PROGRAM prgEM
VAR
	fbKBusState		: FB_K_Bus_State;
	fbEM1			: FB_EM_Beckhoff_KL3403;
	fbEM2			: FB_EM_Beckhoff_KL3403;
	fbEM3			: FB_EM_Beckhoff_KL3403;
	fbEM4			: FB_EM_Beckhoff_KL3403;
	fbEM5			: FB_EM_Beckhoff_KL3403;
	
	wDataL1, wDataL2, wDataL3   AT%I* : WORD;
	bySBL1, bySBL2, bySBL3      AT%I* : BYTE;
	byCBL1, byCBL2, byCBL3      AT%Q*       : BYTE;
	iDataOutL1, iDataOutL2, iDataOutL3  AT%Q* : INT;
	
	fbEM6			: FB_EM_Beckhoff_KL3403;
	fbEM7			: FB_EM_Beckhoff_KL3403;
	fbEM8			: FB_EM_Beckhoff_KL3403;
	fbGrid			: FB_Grid_Power_Ext_Input;			//{#lynus.ag#()}
	lrPowerEM1		: LREAL;							//{#lynus.ag#()}
	lrPowerEM2		: LREAL;							//{#lynus.ag#()}
	lrPowerEM3		: LREAL;							//{#lynus.ag#()}
	lrPowerEM4		: LREAL;							//{#lynus.ag#()}
	lrPowerEM5		: LREAL;							//{#lynus.ag#()}
	lrPowerEM5_1	: LREAL;							//{#lynus.ag#()}
	lrPowerEM5_2	: LREAL;							//{#lynus.ag#()}
	lrPowerEM5_3	: LREAL;							//{#lynus.ag#()}
	lrPowerEM6		: LREAL;							//{#lynus.ag#()}
	lrPowerEM6_1	: LREAL;							//{#lynus.ag#()}
	lrPowerEM6_2	: LREAL;							//{#lynus.ag#()}
	lrPowerEM6_3	: LREAL;							//{#lynus.ag#()}
	lrPowerEM7		: LREAL;							//{#lynus.ag#()}
	lrPowerEM7_1	: LREAL;							//{#lynus.ag#()}
	lrPowerEM7_2	: LREAL;							//{#lynus.ag#()}
	lrPowerEM7_3	: LREAL;							//{#lynus.ag#()}
	lrPowerEM8		: LREAL;							//{#lynus.ag#()}
	lrPowerEM8_1	: LREAL;							//{#lynus.ag#()}
	lrPowerEM8_2	: LREAL;							//{#lynus.ag#()}
	lrPowerEM8_3	: LREAL;							//{#lynus.ag#()}
	lrCounterEM5	: LREAL;							//{#lynus.ag#()}
	lrCounterEM6	: LREAL;							//{#lynus.ag#()}
	lrCounterEM7	: LREAL;							//{#lynus.ag#()}
	lrCounterEM8	: LREAL;							//{#lynus.ag#()}
	
	lrCurrent_EM5_1 : LREAL;							//{#lynus.ag#()}
	lrCurrent_EM5_2 : LREAL;							//{#lynus.ag#()}
	lrCurrent_EM5_3 : LREAL;							//{#lynus.ag#()}
	lrCurrent_EM6_1 : LREAL;							//{#lynus.ag#()}
	lrCurrent_EM6_2 : LREAL;							//{#lynus.ag#()}
	lrCurrent_EM6_3 : LREAL;							//{#lynus.ag#()}
	lrCurrent_EM7_1 : LREAL;							//{#lynus.ag#()}
	lrCurrent_EM7_2 : LREAL;							//{#lynus.ag#()}
	lrCurrent_EM7_3 : LREAL;							//{#lynus.ag#()}
	lrCurrent_EM8_1 : LREAL;							//{#lynus.ag#()}
	lrCurrent_EM8_2 : LREAL;							//{#lynus.ag#()}
	lrCurrent_EM8_3 : LREAL;							//{#lynus.ag#()}
END_VAR

fbKBusState(uiKBusState_OUT=> );


//UV1	
fbEM1(
	bEnable:= TRUE, 
	bChannel1Invers:= TRUE,
	bChannel2Invers:= TRUE,
	bChannel3Invers:= TRUE,
	uiCurrentTransformerRatioL1:= 400, 
	uiCurrentTransformerRatioL2:= 400, 
	uiCurrentTransformerRatioL3:= 400, 
	uiKBusState_IN:= fbKBusState.uiKBusState_OUT, 
	stDataEMPower=> , 
	stDataEMCounter=> , 
	stDataEMPowerRealTime=> , 
	stDataEMCounterRealTime=> , 
	diNrOfEM_OUT=> );

lrPowerEM1 := fbEM1.stDataEMPower.lrPowerTotal;

//UV2	
fbEM2(
	bEnable:= TRUE, 
	bChannel1Invers:= TRUE,
	bChannel2Invers:= TRUE,
	bChannel3Invers:= TRUE,
	uiCurrentTransformerRatioL1:= 400, 
	uiCurrentTransformerRatioL2:= 400, 
	uiCurrentTransformerRatioL3:= 400, 
	uiKBusState_IN:= fbKBusState.uiKBusState_OUT, 
	stDataEMPower=> , 
	stDataEMCounter=> , 
	stDataEMPowerRealTime=> , 
	stDataEMCounterRealTime=> , 
	diNrOfEM_OUT=> );

lrPowerEM2 := fbEM2.stDataEMPower.lrPowerTotal;

//UV3	
fbEM3(
	bEnable:= TRUE, 
	bChannel1Invers:= TRUE,
	bChannel2Invers:= TRUE,
	bChannel3Invers:= TRUE,
	uiCurrentTransformerRatioL1:= 400, 
	uiCurrentTransformerRatioL2:= 400, 
	uiCurrentTransformerRatioL3:= 400, 
	uiKBusState_IN:= fbKBusState.uiKBusState_OUT, 
	stDataEMPower=> , 
	stDataEMCounter=> , 
	stDataEMPowerRealTime=> , 
	stDataEMCounterRealTime=> , 
	diNrOfEM_OUT=> );

lrPowerEM3 := fbEM3.stDataEMPower.lrPowerTotal;	
	
//UV4	
fbEM4(
	bEnable:= TRUE, 
	bChannel1Invers:= TRUE,
	bChannel2Invers:= TRUE,
	bChannel3Invers:= TRUE,
	uiCurrentTransformerRatioL1:= 400, 
	uiCurrentTransformerRatioL2:= 400, 
	uiCurrentTransformerRatioL3:= 400, 
	uiKBusState_IN:= fbKBusState.uiKBusState_OUT, 
	stDataEMPower=> , 
	stDataEMCounter=> , 
	stDataEMPowerRealTime=> , 
	stDataEMCounterRealTime=> , 
	diNrOfEM_OUT=> );

lrPowerEM4 := fbEM4.stDataEMPower.lrPowerTotal;	

//UV5	
fbEM5(
	bEnable:= TRUE, 
	bChannel1Invers:= TRUE,
	bChannel2Invers:= TRUE,
	bChannel3Invers:= TRUE,
	uiCurrentTransformerRatioL1:= 400, 
	uiCurrentTransformerRatioL2:= 400, 
	uiCurrentTransformerRatioL3:= 400, 
	uiKBusState_IN:= fbKBusState.uiKBusState_OUT, 
	stDataEMPower=> , 
	stDataEMCounter=> , 
	stDataEMPowerRealTime=> , 
	stDataEMCounterRealTime=> , 
	diNrOfEM_OUT=> );

lrPowerEM5 := fbEM5.stDataEMPower.lrPowerTotal;	
	lrCounterEM5 := fbEM5.stDataEMCounter.lrTotalCounterEnergy_Consumption;	
		lrPowerEM5_1 := fbEM5.stDataEMPower.lrPowerL1;
			lrPowerEM5_2 := fbEM5.stDataEMPower.lrPowerL2;
				lrPowerEM5_3 := fbEM5.stDataEMPower.lrPowerL3;
					lrCurrent_EM5_1 := fbEM5.stDataEMPower.lrCurrentL1;
						lrCurrent_EM5_2 := fbEM5.stDataEMPower.lrCurrentL2;
							lrCurrent_EM5_3 := fbEM5.stDataEMPower.lrCurrentL3;
	
//UV6
fbEM6(
	bEnable:= TRUE, 
	bChannel1Invers:= TRUE,
	bChannel2Invers:= TRUE,
	bChannel3Invers:= TRUE,
	uiCurrentTransformerRatioL1:= 400, 
	uiCurrentTransformerRatioL2:= 400, 
	uiCurrentTransformerRatioL3:= 400, 
	uiKBusState_IN:= fbKBusState.uiKBusState_OUT, 
	stDataEMPower=> , 
	stDataEMCounter=> , 
	stDataEMPowerRealTime=> , 
	stDataEMCounterRealTime=> , 
	diNrOfEM_OUT=> );

lrPowerEM6 := fbEM6.stDataEMPower.lrPowerTotal;	
	lrCounterEM6 := fbEM6.stDataEMCounter.lrTotalCounterEnergy_Consumption;	
		lrPowerEM6_1 := fbEM6.stDataEMPower.lrPowerL1;
			lrPowerEM6_2 := fbEM6.stDataEMPower.lrPowerL2;
				lrPowerEM6_3 := fbEM6.stDataEMPower.lrPowerL3;
					lrCurrent_EM6_1 := fbEM6.stDataEMPower.lrCurrentL1;
						lrCurrent_EM6_2 := fbEM6.stDataEMPower.lrCurrentL2;
							lrCurrent_EM6_3 := fbEM6.stDataEMPower.lrCurrentL3;
	
//UV7	
fbEM7(
	bEnable:= TRUE, 
	bChannel1Invers:= TRUE,
	bChannel2Invers:= TRUE,
	bChannel3Invers:= TRUE,
	uiCurrentTransformerRatioL1:= 400, 
	uiCurrentTransformerRatioL2:= 400, 
	uiCurrentTransformerRatioL3:= 400, 
	uiKBusState_IN:= fbKBusState.uiKBusState_OUT, 
	stDataEMPower=> , 
	stDataEMCounter=> , 
	stDataEMPowerRealTime=> , 
	stDataEMCounterRealTime=> , 
	diNrOfEM_OUT=> );

lrPowerEM7 := fbEM7.stDataEMPower.lrPowerTotal;
	lrCounterEM7 := fbEM7.stDataEMCounter.lrTotalCounterEnergy_Consumption;	
		lrPowerEM7_1 := fbEM7.stDataEMPower.lrPowerL1;
			lrPowerEM7_2 := fbEM7.stDataEMPower.lrPowerL2;
				lrPowerEM7_3 := fbEM7.stDataEMPower.lrPowerL3;
					lrCurrent_EM7_1 := fbEM7.stDataEMPower.lrCurrentL1;
						lrCurrent_EM7_2 := fbEM7.stDataEMPower.lrCurrentL2;
							lrCurrent_EM7_3 := fbEM7.stDataEMPower.lrCurrentL3;
	
//UV8	
fbEM8(
	bEnable:= TRUE, 
	bChannel1Invers:= TRUE,
	bChannel2Invers:= TRUE,
	bChannel3Invers:= TRUE,
	uiCurrentTransformerRatioL1:= 400, 
	uiCurrentTransformerRatioL2:= 400, 
	uiCurrentTransformerRatioL3:= 400, 
	uiKBusState_IN:= fbKBusState.uiKBusState_OUT, 
	stDataEMPower=> , 
	stDataEMCounter=> , 
	stDataEMPowerRealTime=> , 
	stDataEMCounterRealTime=> , 
	diNrOfEM_OUT=> );

lrPowerEM8 := fbEM8.stDataEMPower.lrPowerTotal;	
	lrCounterEM8 := fbEM8.stDataEMCounter.lrTotalCounterEnergy_Consumption;	
		lrPowerEM8_1 := fbEM8.stDataEMPower.lrPowerL1;
			lrPowerEM8_2 := fbEM8.stDataEMPower.lrPowerL2;
				lrPowerEM8_3 := fbEM8.stDataEMPower.lrPowerL3;
					lrCurrent_EM8_1 := fbEM8.stDataEMPower.lrCurrentL1;
						lrCurrent_EM8_2 := fbEM8.stDataEMPower.lrCurrentL2;
							lrCurrent_EM8_3 := fbEM8.stDataEMPower.lrCurrentL3;
	
//Sum of all 8 Messurements is the Grid power

//Error
IF fbEM5.stDataEMPowerRealTime.byErrorWarning = 2 OR
	fbEM6.stDataEMPowerRealTime.byErrorWarning = 2 OR fbEM7.stDataEMPowerRealTime.byErrorWarning = 2 OR fbEM8.stDataEMPowerRealTime.byErrorWarning = 2 THEN
		fbGrid.bExtErrorGrid := TRUE;
ELSE
		fbGrid.bExtErrorGrid := FALSE;
END_IF	

//Power and Counter Data
fbGrid.lrExtGridPower := fbEM5.stDataEMPowerRealTime.lrPowerTotal +
							fbEM6.stDataEMPowerRealTime.lrPowerTotal + fbEM7.stDataEMPowerRealTime.lrPowerTotal + fbEM8.stDataEMPowerRealTime.lrPowerTotal;

fbGrid.lrExtCounterEnergyT1_Consumption := fbEM5.stDataEMCounterRealTime.lrCounterEnergyT1_Consumption + fbEM6.stDataEMCounterRealTime.lrCounterEnergyT1_Consumption +
													fbEM7.stDataEMCounterRealTime.lrCounterEnergyT1_Consumption + fbEM8.stDataEMCounterRealTime.lrCounterEnergyT1_Consumption;	

fbGrid.lrExtCounterEnergyT2_Consumption := fbEM5.stDataEMCounterRealTime.lrCounterEnergyT2_Consumption + fbEM6.stDataEMCounterRealTime.lrCounterEnergyT2_Consumption +
													fbEM7.stDataEMCounterRealTime.lrCounterEnergyT2_Consumption + fbEM8.stDataEMCounterRealTime.lrCounterEnergyT2_Consumption;							
							
fbGrid.lrExtTotalCounterEnergy_Consumption := fbEM5.stDataEMCounterRealTime.lrTotalCounterEnergy_Consumption + fbEM6.stDataEMCounterRealTime.lrTotalCounterEnergy_Consumption +
													fbEM7.stDataEMCounterRealTime.lrTotalCounterEnergy_Consumption + fbEM8.stDataEMCounterRealTime.lrTotalCounterEnergy_Consumption;
													
fbGrid.lrExtCounterEnergyT1_Production := fbEM5.stDataEMCounterRealTime.lrCounterEnergyT1_Production + fbEM6.stDataEMCounterRealTime.lrCounterEnergyT1_Production +
													fbEM7.stDataEMCounterRealTime.lrCounterEnergyT1_Production + fbEM8.stDataEMCounterRealTime.lrCounterEnergyT1_Production; 
													
fbGrid.lrExtCounterEnergyT2_Production := fbEM5.stDataEMCounterRealTime.lrCounterEnergyT2_Production + fbEM6.stDataEMCounterRealTime.lrCounterEnergyT2_Production +
													fbEM7.stDataEMCounterRealTime.lrCounterEnergyT2_Production + fbEM8.stDataEMCounterRealTime.lrCounterEnergyT2_Production; 
													
fbGrid.lrExtTotalCounterEnergy_Production := fbEM5.stDataEMCounterRealTime.lrTotalCounterEnergy_Production + fbEM6.stDataEMCounterRealTime.lrTotalCounterEnergy_Production +
													fbEM7.stDataEMCounterRealTime.lrTotalCounterEnergy_Production + fbEM8.stDataEMCounterRealTime.lrTotalCounterEnergy_Production;

fbGrid(
	bEnable:= TRUE, 
	diNrOfEMS_IN:= 1, 
	rSizeGridConn:= , 
	bExtErrorGrid:= , 
	lrExtGridPower:= , 
	lrExtTotalCounterEnergy_Consumption:= , 
	lrExtTotalCounterEnergy_Production:= , 
	lrExtCounterEnergyT1_Consumption:= , 
	lrExtCounterEnergyT2_Consumption:= , 
	lrExtCounterEnergyT1_Production:= , 
	lrExtCounterEnergyT2_Production:= , 
	stDataGrid=> , 
	diNrOfGrid_OUT=> );

END_PROGRAM

(* stored: Version 1.1.0.1, ProductVersion 3.1.4024.9
   POU prgEM: Id {1c0bba27-fd31-45cc-b497-003c89abb689}, SpecialFunc None *)
